INTERFACE I_ServerResponseConfig

METHOD PUBLIC UpdateResponseWithAccepted
VAR_INPUT
	Response : I_ServerResponse;
END_VAR
END_METHOD

METHOD PUBLIC UpdateResponseWithBusy
VAR_INPUT
	Response : I_ServerResponse;
END_VAR
END_METHOD

METHOD PUBLIC UpdateResponseWithError
VAR_INPUT
	Response : I_ServerResponse;
	Message : T_MAXSTRING;
END_VAR
END_METHOD

METHOD PUBLIC UpdateResponseWithPending
VAR_INPUT
	Response : I_ServerResponse;
	ResponseId : T_MAXSTRING;
	RetryDelayInMs : UDINT;
END_VAR
END_METHOD

METHOD PUBLIC UpdateResponseWithSuccess
VAR_INPUT
	Response : I_ServerResponse;
END_VAR
END_METHOD

END_INTERFACE

(* stored: Version 1.1.0.1, ProductVersion 3.1.4024.12
   Itf I_ServerResponseConfig: Id {7bbdf4b5-2dfc-4158-a62c-7ac7f8bed0f1}
   Method UpdateResponseWithAccepted: Id {55682826-e6fd-4c15-adc0-0d952235138a}
   Method UpdateResponseWithBusy: Id {a95a1314-fcdc-4872-addf-8a57f65f0cb1}
   Method UpdateResponseWithError: Id {b0641bf5-c983-49ae-9619-021c434d7cc3}
   Method UpdateResponseWithPending: Id {759d8788-6614-465c-a216-be4f17d1937b}
   Method UpdateResponseWithSuccess: Id {e484e660-a1f7-41de-83b0-02ff4fd45376} *)
